// TwinCAT 3 PLC project TcLog
// Title: TcLog
// Company: Benedikt Geisler
// Author: Benedikt Geisler
// ProjectVersion: 0.6.1
// Description: TcLog provides logging functionality to TwinCAT.
// ProgramVersion: 3.1.4026.20
// libraries:
//   Tc2_Standard, * (Beckhoff Automation GmbH)
//   Tc2_System, * (Beckhoff Automation GmbH)
//   Tc2_Utilities, * (Beckhoff Automation GmbH)
//   Tc3_DynamicMemory, * (Beckhoff Automation GmbH)
// project tree:
//   / Constants.TcGVL (not stored)
//   Logger/DataTypes/ Error.TcDUT, ErrorCodes.TcDUT, LoggingConfiguration.TcDUT (not stored), LogLevels.TcDUT (not stored), RollingIntervals.TcDUT
//   Logger/Interfaces/ ILog.TcIO, ILogCore.TcIO
//   Logger/ LogLevelToAdsLogMsgType.TcPOU (not stored), TcLog.TcPOU (not stored), TcLogCore.TcPOU, TcLogTrig.TcPOU
//   StringBuilder/Interfaces/ ILimitedStringBuilder.TcIO (not stored), IStringBuilder.TcIO (not stored)
//   StringBuilder/ StringBuilder.TcPOU (not stored)
//   Utils/ AnyToString.TcPOU (not stored), DateTime.TcPOU, DeleteOldFiles.TcPOU (not stored), DynamicStringBuffer.TcPOU, GetFileAgeInSeconds.TcPOU (not stored)
//   Utils/DataTypes/ DeleteFilesState.TcDUT (not stored), PersistToFileState.TcDUT (not stored)

// ---- Logger/DataTypes/Error.TcDUT
/// This is the error type used in this library.
TYPE Error :
STRUCT
  /// `TRUE` signals an active error
	Active : BOOL;
  /// Error code of type `ErrorCodes`
	Code : INT;
  /// Plain text error message
	Info : Tc2_System.T_MaxString;
END_STRUCT
END_TYPE

// ---- Logger/DataTypes/ErrorCodes.TcDUT
/// Provides error codes for TcLogCore
{attribute 'qualified_only'}
{attribute 'strict'}
{attribute 'to_string'}
TYPE ErrorCodes : 
(
	None := 0,
	OpeningFileFailed,
	WritingToFileFailed,
	ClosingFileFailed,
	EnumeratingFilesInSpecifiedDirectoryFailed,
	DeletingFileFailed,
	FifoOverflow
);
END_TYPE

// ---- Logger/DataTypes/RollingIntervals.TcDUT
/// Rolling interval to create a new log file when expired. 
{attribute 'qualified_only'}
{attribute 'strict'}
{attrivute 'to_string'}
TYPE RollingIntervals :
(
	None := 0,
	Hourly,
	Daily,
	Monthly
);
END_TYPE

// ---- Logger/Interfaces/ILog.TcIO
INTERFACE PUBLIC ILog

METHOD SetLogger : BOOL
VAR_INPUT
    ref2Core : ILogCore;
END_VAR
END_METHOD

END_INTERFACE

// ---- Logger/Interfaces/ILogCore.TcIO
INTERFACE PUBLIC ILogCore EXTENDS __SYSTEM.IQueryInterface

// Logger method.
// Logs data in custom format. No additional formatting will be done.
METHOD LogCustomFormat : BOOL
VAR_INPUT
    data : Tc2_System.T_MaxString; // Data to be logged. No additional formatting will be done.
END_VAR
END_METHOD

// Logger method.
// Logs in the standard format. This includes
// - timestamp
// - log level
// - log message
// - instance path of logging source (optional)
// The message will only be logged if the logging level exceeds the configured minimum logging level.
METHOD LogStandardFormat : BOOL
VAR_INPUT
    data : Tc2_System.T_MaxString; // Data to be logged. Additional formatting wil be done.
    instancePath : Tc2_System.T_MaxString; // Instance path of calling logger to locate source of logging message.
    logLevel : LogLevels; // Log level of message.
END_VAR
END_METHOD

END_INTERFACE

// ---- Logger/TcLogCore.TcPOU
/// `TcLogCore` provides the base functionality of the logger and sets the configuration.
/// The logger can be configured by calling its methods that set the configuration.
///
/// > [!NOTE]
/// > `TcLogCore.RunLogger()` should be called once each cycle. The configuration methods should be called **before** 
/// > `RunLogger` is called.
///
/// When declaring an instance of TcLogCore, the ininital buffer size has to be set. If the buffer size is set too low, it will expand
/// automatically if enough memory is available.
///
/// To set the inital buffer size to accomodate 100 messages, use it like this:
///
/// ```st
/// VAR
///   myLogger: TcLogCore(BufferSize := 100 * (Tc2_System.MAX_STRING_LENGTH * Constants.FifoOverhead));
/// END_VAR
/// ```
///
{attribute 'linkalways'}
{attribute 'hide_all_locals'}
FUNCTION_BLOCK PUBLIC TcLogCore IMPLEMENTS ILogCore
VAR
	_loggingSingleton : TcLog; // Logger-Singleton: Required to provide Singleton-functionality for TcLog.
	_utcTimeAsFileTime : Tc2_Utilities.T_FILETIME; // Current utc time as filetime
	_localTimeAsSystemTime : Tc2_Utilities.TIMESTRUCT; // Current local time as timestring
	_localTimeAsString : STRING; // Current local time as string
	_logCache : DynamicStringBuffer; // Dynamic string buffer to cache logs to be processed
	_startLoggingConfiguration : BOOL; // Aux variable to provide fluent interface.
	_internalErrorOccured : BOOL; // Aux variable to log internal errors to Error-property.                                                   				
	_config : LoggingConfiguration; // Logging configuration. Is set by invoking configuration methods.
	_error : Error; // Contains information about internal error.
	_busy : BOOL; // Logger is busy, typically with writing logs to the file system.
  _timeInfoReady : BOOL := FALSE; // Set to true once the time information is available
END_VAR

// Nothing to be done here. Logger works by invoking its methods.
// "RunLogger" contains all the implementation that has to be processed cyclically.

// Builds logging configuration.
// Required to provide a fluent interface.
// Has to be called at the begin of each method that configures the logger.
{attribute 'hide'}
METHOD PRIVATE BuildLoggingConfiguration : BOOL
IF NOT _startLoggingConfiguration THEN
	_startLoggingConfiguration := TRUE;
	
	_config.RollingInterval := RollingIntervals.Daily;
	_config.WriteToAds := FALSE;
	_config.FileName := '';
	_config.FilePath := 'c:\';
	_config.MinimumLevel := LogLevels.Debug;
	_config.Delimiter := '|';
	_config.IncludeInstancePath := FALSE;
	_config.LogFileLifespan := 0;
	_config.TimestampFormat := 'YYYYMMDD_hhmm_';
	_config.ValidTimestampsOnly := FALSE;
END_IF
END_METHOD

/// `Busy` evaluates to `TRUE` as long as the log file is kept open to append new log messages
/// or there are pending messages in the queue to be written to the logfile.
{attribute 'monitoring':='call'}
PROPERTY Busy : BOOL
GET
Busy := _busy;
END_GET
SET // PRIVATE
_busy := Busy;
END_SET
END_PROPERTY

/// Returns the current configuration of the logger.
{attribute 'monitoring':='variable'}
PROPERTY Configuration : LoggingConfiguration
GET
Configuration := _config;
END_GET
END_PROPERTY

/// Configuration method which sets the lifespan of log files. Once exceeded, they will be deleted.
METHOD DeleteLogFilesAfterDays : REFERENCE TO TcLogCore
VAR_INPUT
  /// Lifespan of logfiles in days.
	lifespan : UINT; 
END_VAR
BuildLoggingConfiguration();

_config.LogFileLifespan := lifespan;

DeleteLogFilesAfterDays REF= THIS^;
END_METHOD

/// Returns information about internal errors.
{attribute 'monitoring':='call'}
{attribute 'suppress_wrn_C0410'}
PROPERTY Error : REFERENCE TO Error
GET
Error REF= _error;
END_GET
END_PROPERTY

METHOD FB_init : BOOL
VAR_INPUT
	bInitRetains : BOOL; // if TRUE, the retain variables are initialized (warm start / cold start)
	bInCopyCode : BOOL; // if TRUE, the instance afterwards gets moved into the copy code (online change)
  /// Initial buffer size for the internal log message buffer
	bufferSize : UDINT;
END_VAR
_loggingSingleton.Init(THIS^);
_logCache.Init(bufferSize);
END_METHOD

/// Flushes the logging cache. All messages that have not yet been processed will be lost.
METHOD FlushCache : BOOL
_logCache.FlushCache();
END_METHOD

/// Configuration method. If this method is called, the instance path where the log 
/// messages has been triggered will be included in the log message. 
METHOD IncludeInstancePath : REFERENCE TO TcLogCore
BuildLoggingConfiguration();

_config.IncludeInstancePath := TRUE;

IncludeInstancePath REF= This^;
END_METHOD

/// Logger method. It should only be called from within objects that implement `ILog`.
/// Logs data in custom format. No additional formatting will be done. 
METHOD LogCustomFormat : BOOL
VAR_INPUT
  /// Data to be logged.
	data : Tc2_System.T_MaxString; 
END_VAR
IF(TimeInfoReady OR NOT _config.ValidTimestampsOnly) THEN 
	IF _config.WriteToAds THEN 
		Tc2_System.ADSLOGSTR(ADSLOG_MSGTYPE_LOG OR ADSLOG_MSGTYPE_HINT, data, ''); 
	END_IF
	
	IF _config.FileName <> '' THEN 
		_logCache.AddLine(data);
	END_IF
END_IF
END_METHOD

/// Logger method. It should only be called from within objects that implement `ILog`.
/// Logs in the standard format. This includes
/// - timestamp
/// - log level
/// - log message
/// - instance path of logging source (optional)
/// The message will only be logged if the logging level exceeds the configured minimum logging level.
METHOD LogStandardFormat : BOOL
VAR_INPUT
  /// Data to be logged.
	data : Tc2_System.T_MaxString; 
  /// Instance path of calling logger to locate source of logging message.
	instancePath : Tc2_System.T_MaxString;
  /// Log level of message. 
	logLevel : LogLevels; 
END_VAR
VAR_INST
  {attribute 'hide'}
	messageBuilder : StringBuilder;
END_VAR
IF LogLevel >= _config.MinimumLevel AND (TimeInfoReady OR NOT _config.ValidTimestampsOnly)  THEN
	IF _config.WriteToAds THEN 
		Tc2_System.ADSLOGSTR(
			ADSLOG_MSGTYPE_LOG OR LogLevelToAdsLogMsgType(logLevel), 
			messageBuilder
				.Reset()
				.AppendIf(_config.IncludeInstancePath, instancePath)
				.AppendIf(_config.IncludeInstancePath, _config.Delimiter)
				.Append(data)
				.ToString(), 
			''
		); 
	END_IF
	
	IF _config.FileName <> '' THEN 
		_logCache.AddLine(
			messageBuilder
					.Reset()
					.Append(_localTimeAsString)
					.Append(_config.Delimiter)
					.Append(TO_STRING(LogLevel))
					.AppendIf(_config.IncludeInstancePath, _config.Delimiter)
					.AppendIf(_config.IncludeInstancePath, instancePath)
					.Append(_config.Delimiter)
					.Append(data)
					.ToString()
		);
	END_IF
END_IF
END_METHOD

/// Configuration method.
/// Sets the minimum log level. Log messages below this level 
/// will not be logged.
METHOD MinimumLevel : REFERENCE TO TcLogCore
VAR_INPUT
  /// Minimum log level to be logged.
	level : LogLevels; 
END_VAR
BuildLoggingConfiguration();

_config.MinimumLevel := level;

MinimumLevel REF=THIS^;
END_METHOD

// Checks the specified rolling interval for the file name.
// Generates new file name if rolling intervall exceeded.
{attribute 'hide_all_locals'}
{attribute 'hide'}
METHOD PRIVATE RollingIntervalReached : BOOL
VAR_INPUT
	currentUtcTime : Tc2_Utilities.TIMESTRUCT;  // Current system time as utc
	rollingInterval : RollingIntervals; // Rolling interval 
END_VAR
VAR_INST
	newHour : Tc2_Standard.R_TRIG;
	newDay : Tc2_Standard.R_TRIG;
	newMonth : Tc2_Standard.R_TRIG;
	
	hourRolled : BOOL;
	dayRolled : BOOL;
	monthRolled : BOOL;
END_VAR
newHour(CLK := (currentUtcTime.wMinute = 0 AND currentUtcTime.wSecond = 0), 
	Q => hourRolled);
newDay(CLK := (hourRolled AND currentUtcTime.wHour = 0), 
	Q => dayRolled);
newMonth(CLK := (dayRolled AND currentUtcTime.wDay = 1), 
	Q => monthRolled);

RollingIntervalReached := 	(hourRolled 	AND rollingInterval = RollingIntervals.Hourly) OR
							(dayRolled 		AND rollingInterval = RollingIntervals.Daily) 	OR
							(monthRolled 	AND rollingInterval = RollingIntervals.Monthly);
END_METHOD

/// Cyclic method of Logger.
/// This method has to be executed in every plc cycle and runs 
/// all internal methods that have to be executed cyclically.
/// > [!NOTE]
/// > This method should be the last method of `TcLogCore` to be called in each cycle.
{attribute 'hide_all_locals'}
METHOD RunLogger : BOOL
VAR_INST
	newDay : Tc2_Standard.R_TRIG; 
	dateTime : DateTime;
	deleteExpiredLogFiles : DeleteOldFiles;
	fileNameStringBuilder : StringBuilder;
	timeStamp : STRING; // Timestamp used for filename
END_VAR
// Generate time data (shared state)
dateTime();
IF dateTime.Done THEN _timeInfoReady := TRUE; END_IF

_localTimeAsSystemTime := dateTime.AsLocalSystemTime;
_localTimeAsString := dateTime.AsLocalSystemTimeString;
_utcTimeAsFileTime := dateTime.AsUtcFileTime;

// Generate new timestamp for filename
IF RollingIntervalReached(_localTimeAsSystemTime, _config.RollingInterval) OR dateTime.Done THEN
	timeStamp := dateTime.ToFormatString(_config.TimestampFormat);
END_IF

// Delete expired log files
newDay(CLK := _localTimeAsSystemTime.wHour = 0);
deleteExpiredLogFiles(
	StartScan 			:= 	newDay.Q AND (_config.LogFileLifespan > 0),
	ExpirationInDays 	:=	_config.LogFileLifespan,
	FilePath			:=	_config.FilePath,
	FileName 			:=	_config.FileName,
	CurrentUtcTime 		:= 	_utcTimeAsFileTime	
	);
IF deleteExpiredLogFiles.Error.Active THEN
	_internalErrorOccured := TRUE;
	_error := deleteExpiredLogFiles.Error;
END_IF
		
// Persist logging messages to file
_logCache.PersistToFile(
  TimeInfoReady,
	fileNameStringBuilder
		.Reset()
		.Append(_config.FilePath)
		.AppendIf(Tc2_Standard.RIGHT(_config.FilePath, 1) <> '\', '\')
		.Append(timeStamp)
		.Append(_config.FileName)
		.ToString()
);
IF _logCache.Error.Active THEN
	_internalErrorOccured := TRUE;
	_error := _logCache.Error;
END_IF

// Forward busy state of LogCache 
Busy := _logCache.Busy;

// Reset Logging configuration: neccesary in order to provide fluent interface
_startLoggingConfiguration := FALSE;

// Reset error flag each cycle to automatically confirm errors once they are gone.
IF NOT _internalErrorOccured THEN
	_error.Active := FALSE;
	_error.Code := ErrorCodes.None;
	_error.Info := '';
END_IF
_internalErrorOccured := FALSE;
END_METHOD

/// Configuration method
/// Sets delimiter between different columns of log file.
METHOD SetDelimiter : REFERENCE TO TcLogCore
VAR_INPUT
  /// Delimiter between different columns of log file.
	delimiter : STRING(1); 
END_VAR
BuildLoggingConfiguration();

_config.Delimiter := delimiter;

SetDelimiter REF=THIS^;
END_METHOD

/// Configuration method.
/// Sets the rolling interval of the log file. Once the rolling interval
/// expires, a file name with a new timestamp will be generated.
METHOD SetRollingInterval : REFERENCE TO TcLogCore
VAR_INPUT
  /// Rolling interval for log file. Once exceeded, a new log file will be created.
	interval : RollingIntervals; 
END_VAR
BuildLoggingConfiguration();

_config.RollingInterval := interval;

SetRollingInterval REF= THIS^;
END_METHOD

/// `TimeInfoReady` evaluates to `TRUE` once the time information used by determine
/// the timestamp for the message is available.
{attribute 'monitoring':='call'}
PROPERTY TimeInfoReady : BOOL
GET
TimeInfoReady := _timeInfoReady;
END_GET
END_PROPERTY

/// Configuration method.
/// Sets the format of the timestamp in the file name. 
/// 
/// The following format options are available:
///	Y : year
///	M : month
/// D : day
/// h : hour 
/// m : minute
/// s : second
/// i : millisecond
/// 
/// Example: _YYMMDD-hh:mm:ss:iii_
/// => _20210812-12:30:22:123_
METHOD TimestampFormat : REFERENCE TO TcLogCore
VAR_INPUT
  /// Format the timestamp should have.
	format : STRING; 
END_VAR
BuildLoggingConfiguration();

_config.TimestampFormat := format;

TimestampFormat REF= THIS^;
END_METHOD

/// Configuration method. If this method is called, only valid timestamps are logged.
/// Note that using this configuration will skip logging anything during the first few PLC cycles, 
/// as TwinCAT needs a few cycles to initialize its time information.
METHOD ValidTimestampsOnly : REFERENCE TO TcLogCore
BuildLoggingConfiguration();

_config.ValidTimestampsOnly := TRUE;

ValidTimestampsOnly REF= This^;
END_METHOD

/// Configuration method.
/// If this method is called, the logs will be written to ADS.
METHOD WriteToAds : REFERENCE TO TcLogCore
BuildLoggingConfiguration();

_config.WriteToAds := TRUE;

WriteToAds REF= This^;
END_METHOD

/// Configuration method.
/// If this method is called, the logs will be persisted to the file system.
METHOD WriteToFile : REFERENCE TO TcLogCore
VAR_INPUT
  /// File path the logs will be written to.
	path : Tc2_System.T_MaxString; 
  /// File name of the log file. Will automatically be prefixed by timestamp.
	fileName : STRING; 
END_VAR
BuildLoggingConfiguration();

IF Tc2_Standard.RIGHT(path, 1) <> '\' THEN
  _config.FilePath := TC2_Standard.CONCAT(path, '\');  
ELSE
  _config.FilePath := path;
END_IF
_config.FileName := fileName;

WriteToFile REF= This^;
END_METHOD

END_FUNCTION_BLOCK

// ---- Utils/DynamicStringBuffer.TcPOU
{attribute 'hide_all_locals'}
FUNCTION_BLOCK INTERNAL DynamicStringBuffer
VAR_OUTPUT
  Error : Error; // Error information of this FB
END_VAR
VAR
  _fifo : Tc2_Utilities.FB_StringRingBuffer; // Necessary to buffer log data until it has been written to file.
  _memoryManager : Tc3_DynamicMemory.FB_DynMem_Manager; // Memory manager, required by DynMem_Buffer.
  _dynamicMemoryBuffer : Tc3_DynamicMemory.FB_DynMem_Buffer(ipMemMan := _memoryManager); // Provides dynamic buffer for Fifo. Is extended automatically if more than the
                                                                   // default buffer size is needed.                  
  _busy : BOOL; // Buffer is busy; typically with writing data to the file system.
END_VAR

METHOD AddLine : BOOL
VAR_INPUT
  text : Tc2_System.T_MaxString; // Text to be added to the buffer
END_VAR
ResizeFifoBufferIfNecessary();
_fifo.A_AddTail(putValue := Tc2_Standard.CONCAT(Tc2_Standard.LEFT(text, 254), '$N'));
END_METHOD

METHOD AddString : BOOL
VAR_INPUT
  text : Tc2_System.T_MaxString; // String to be added to the buffer
END_VAR
ResizeFifoBufferIfNecessary();
_fifo.A_AddTail(putValue := text);
END_METHOD

METHOD PRIVATE AllocateBuffer : BOOL // Allocates buffer FOR the fifo.
VAR_INPUT
  bufferSize : UDINT; // Initial buffer size in BYTEs for fifo buffer.
END_VAR
_dynamicMemoryBuffer.CreateBuffer(nSize:=bufferSize, bReset:=TRUE);
_fifo.pBuffer := _dynamicMemoryBuffer.pBuffer;
_fifo.cbBuffer := bufferSize;
END_METHOD

{attribute 'monitoring':='call'}
PROPERTY Busy : BOOL
GET
Busy := _busy;
END_GET
SET // PRIVATE
_busy := Busy;
END_SET
END_PROPERTY

METHOD FB_exit : BOOL
VAR_INPUT
  bInCopyCode : BOOL; // if TRUE, the exit method is called for exiting an instance that is copied afterwards (online change).
END_VAR
_dynamicMemoryBuffer.Clear();
END_METHOD

METHOD FlushCache : BOOL
_fifo.A_Reset();
END_METHOD

METHOD INTERNAL Init : BOOL
VAR_INPUT
  bufferSize : UDINT; // Initial buffer size in BYTEs for fifo buffer.
END_VAR
AllocateBuffer(bufferSize);
END_METHOD

{attribute 'hide_all_locals'}
METHOD PersistToFile : BOOL
VAR_INPUT
  enable: BOOL; // TRUE starts persistence mechanism
  fileName : Tc2_System.T_MaxString; // File name including its path
END_VAR
VAR_INST
  state : PersistToFileState;
  
  fileOpen : Tc2_System.FB_FileOpen;
  fileHandle : UINT;
  
  fileWrite : Tc2_System.FB_FileWrite;
  lockFileWriteToForceRisingEdge : BOOL; // filePuts can only be executed every other cycle
                                         // since it needs a rising edge to execute.
  fileClose : Tc2_System.FB_FileClose;
  
  buffer : ARRAY[0..CONSTANTS.BufferSize] OF BYTE;
  currentBufferPos : UDINT;
  fifoHeadString : Tc2_System.T_MaxString;
  fifoHeadLength : UDINT;
  fifoHeadBytes : ARRAY[0..Tc2_System.MAX_STRING_LENGTH] OF BYTE;
  i : UINT;
END_VAR
VAR CONSTANT
  NetId : STRING := '';
  Timeout : TIME := DEFAULT_ADS_TIMEOUT;
  MaxLogsPerCycle : UINT := UDINT_TO_UINT(CONSTANTS.BufferSize / Tc2_System.MAX_STRING_LENGTH);
  MaxBufferPosition : UDINT := (SIZEOF(buffer)-Tc2_System.MAX_STRING_LENGTH);
END_VAR
// State machine
// Using if-statements instead of case for performance reasons:
// Some states execute instantly and allow thus the next state 
// to start within the same plc cycle.

// *** I D L E ***
IF state = PersistToFileState.Idle THEN
  lockFileWriteToForceRisingEdge := FALSE;
  IF _fifo.nCount > 0 AND enable THEN 
    lockFileWriteToForceRisingEdge := FALSE;
    state := PersistToFileState.OpenFile;
  END_IF
END_IF
    
// *** O P E N   F I L E ***
fileOpen(sNetId := NetId, sPathName := fileName, nMode := FOPEN_MODEAPPEND OR FOPEN_MODETEXT, 
           ePath := PATH_GENERIC, bExecute := (state = PersistToFileState.OpenFile), tTimeout := Timeout,
           hFile => fileHandle);

IF state = PersistToFileState.OpenFile THEN
  IF fileOpen.bError THEN
    state := PersistToFileState.CloseFile;
  ELSIF NOT fileOpen.bBusy THEN
    state := PersistToFileState.GetStringFromFifo; 
  END_IF
END_IF 

// *** P O P   F R O M   F I F O ***
IF state = PersistToFileState.GetStringFromFifo THEN
  IF NOT lockFileWriteToForceRisingEdge THEN
    currentBufferPos := 0;
    FOR i:=0 TO MaxLogsPerCycle DO
      IF _fifo.nCount <= 0 THEN EXIT; END_IF
      IF currentBufferPos >= MaxBufferPosition THEN EXIT; END_IF
      
      _fifo.A_RemoveHead(getValue => fifoHeadString); 
      fifoHeadBytes := MAXSTRING_TO_BYTEARR(fifoHeadString);
      fifoHeadLength := INT_TO_UDINT(LEN(fifoHeadString));
      MEMCPY(
        destAddr  :=  ADR(buffer) + SIZEOF(BYTE) * currentBufferPos,
        srcAddr   :=  ADR(fifoHeadBytes),
        n     :=  fifoHeadLength);    
      currentBufferPos := currentBufferPos + fifoHeadLength;  
    END_FOR
    state := PersistToFileState.AppendDataToFile;
  END_IF
  lockFileWriteToForceRisingEdge := FALSE;
END_IF
  
// *** W R I T E   T O   F I L E ***
fileWrite(
  sNetId := NetId, 
  hFile := fileHandle, 
  pWriteBuff := ADR(buffer),
  cbWriteLen := currentBufferPos,
  bExecute := state = PersistToFileState.AppendDataToFile, 
  tTimeout := Timeout); 

IF state = PersistToFileState.AppendDataToFile THEN
  lockFileWriteToForceRisingEdge := TRUE;   
  IF fileWrite.bError THEN
    state := PersistToFileState.CloseFile;
  ELSIF _fifo.nCount > 0 AND NOT fileWrite.bBusy THEN
    state := PersistToFileState.GetStringFromFifo; 
  ELSIF _fifo.nCount = 0 THEN
    state := PersistToFileState.CloseFile;
  END_IF
END_IF
    
// *** C L O S E   F I L E ***
fileClose(
  sNetId := NetId, hFile := fileHandle, 
  bExecute := (state = PersistToFileState.CloseFile), tTimeout := Timeout);

IF state = PersistToFileState.CloseFile THEN
  IF NOT fileClose.bBusy THEN state := PersistToFileState.Idle; END_IF
END_IF

// Close file in case of error
IF fileOpen.bError THEN state := PersistToFileState.CloseFile; END_IF
IF fileWrite.bError THEN state := PersistToFileState.CloseFile; END_IF
IF NOT _fifo.bOk AND _fifo.nCount > 0 AND state <> PersistToFileState.Idle THEN 
  state := PersistToFileState.CloseFile; 
END_IF

// Error handling
IF fileOpen.bError THEN
  Error.Active := TRUE;
  Error.Code := ErrorCodes.OpeningFileFailed;
  Error.Info := Tc2_Standard.CONCAT('Opening file failed. Error thrown by FB_FileOpen. Consult Beckhoff InfoSys. Internal Error: ', UDINT_TO_STRING(fileOpen.nErrId));
ELSIF fileWrite.bError THEN
  Error.Active := TRUE;
  Error.Code := ErrorCodes.WritingToFileFailed;
  Error.Info := Tc2_Standard.CONCAT('Writing to file failed. Error thrown by FB_FileWrite. Consult Beckhoff InfoSys. Internal Error: ', UDINT_TO_STRING(fileWrite.nErrId));
ELSIF fileClose.bError THEN
  Error.Active := TRUE;
  Error.Code := ErrorCodes.ClosingFileFailed;
  Error.Info := Tc2_Standard.CONCAT('Closing file failed. Error thrown by FB_FileClose. Consult Beckhoff InfoSys. Internal Error: ', UDINT_TO_STRING(fileClose.nErrId));
ELSIF NOT _fifo.bOk AND _fifo.nCount > 0 THEN
  Error.Active := TRUE;
  Error.Code := ErrorCodes.FifoOverflow;
  Error.Info := 'FIFO overflow. Check if plc has enough free memory.';
ELSE
  Error.Active := FALSE;
  Error.Code := ErrorCodes.None;
  Error.Info := '';
END_IF

// Set busy state
Busy := (state <> PersistToFileState.Idle OR _fifo.nCount > 0);

(* Uncomment for cyclic logging of state machine, buffer usage & errors

ADSLOGSTR(ADSLOG_MSGTYPE_LOG, 
  Tc2_Standard.CONCAT('****DynamicStringBuffer.state:', 
  Tc2_Standard.CONCAT(UINT_TO_STRING(state),
  Tc2_Standard.CONCAT(', DynamicStringBuffer.hFile:', UINT_TO_STRING(hFile)))), '');

ADSLOGSTR(ADSLOG_MSGTYPE_LOG, 
  Tc2_Standard.CONCAT('****Fifo: used ', 
  Tc2_Standard.CONCAT(UDINT_TO_STRING(Fifo.cbSize),
  Tc2_Standard.CONCAT(' of ', UDINT_TO_STRING(Fifo.cbBuffer)))), '');
  
IF Error.Active THEN
  ADSLOGSTR(ADSLOG_MSGTYPE_LOG, 
    Tc2_Standard.CONCAT('****DynamicStringBuffer.Error: ', Error.Info), 
    '');  
END_IF
*)
END_METHOD

METHOD PopHead : Tc2_System.T_MaxString
VAR_INST
  headString : Tc2_System.T_MaxString;
END_VAR
_fifo.A_RemoveHead(getValue => headString);
PopHead := headString;
END_METHOD

// Resizes the buffer for the FIFO if necessary
METHOD PRIVATE ResizeFifoBufferIfNecessary : BOOL
VAR
  requiredSize : UDINT;
  newSize : DINT;
END_VAR
requiredSize := _fifo.cbSize + (Tc2_System.MAX_STRING_LENGTH + Constants.FifoOverhead);

IF requiredSize > _fifo.cbBuffer THEN
  _dynamicMemoryBuffer.Resize(nSize := requiredSize*SIZEOF(BYTE), bPreserve:=TRUE, bReset:=TRUE);
  _fifo.pBuffer := _dynamicMemoryBuffer.pBuffer;
  _fifo.cbBuffer := requiredSize;
END_IF
END_METHOD

END_FUNCTION_BLOCK

// ---- Utils/DateTime.TcPOU
/// Generate time data in different formats.
{attribute: 'hide_all_locals'}
FUNCTION_BLOCK DateTime
VAR
  _localSystemTime : Tc2_Utilities.FB_LocalSystemTime;
  _getSystemTime : Tc2_System.GETSYSTEMTIME;
  _timeZoneInfo : Tc2_Utilities.FB_GetTimeZoneInformation;
  _localTime : Tc2_Utilities.FB_SystemTimeToTzSpecificLocalTime;
  _localSystemTimeValid : Tc2_Standard.R_TRIG;
  _utcTime : Tc2_Utilities.FB_TzSpecificLocalTimeToFileTime;
END_VAR

// Get local system time
_localSystemTime(
  sNetID  :=  '',
  bEnable :=  TRUE,
  dwCycle :=  1,
  dwOpt :=  1,
  tTimeout:=  DEFAULT_ADS_TIMEOUT
);

// Get timezone information
_timeZoneInfo(
  sNetID := '',
  bExecute := TRUE,
  tTimeout := DEFAULT_ADS_TIMEOUT);

// Convert local time to utc time
_utcTime(
  in := THIS^.AsLocalFileTime,
  tzInfo := _timeZoneInfo.tzInfo);
  
// Finished retrieving time data
_localSystemTimeValid(CLK := _localSystemTime.bValid);

/// Returns local time as `Tc2_Utilities.T_FILETIME`.
{attribute 'monitoring':='variable'}
PROPERTY AsLocalFileTime : Tc2_Utilities.T_FILETIME
GET
AsLocalFileTime := SYSTEMTIME_TO_FILETIME(THIS^.AsLocalSystemTime);
END_GET
END_PROPERTY

/// Returns local time as `Tc2_Utilities.TIMESTRUCT`.
{attribute 'monitoring':='variable'}
PROPERTY AsLocalSystemTime : Tc2_Utilities.TIMESTRUCT
GET
AsLocalSystemTime := _localSystemTime.systemTime;
END_GET
END_PROPERTY

/// Returns local time as string.
{attribute 'monitoring':='variable'}
PROPERTY AsLocalSystemTimeString : Tc2_System.T_MAXSTRING
GET
AsLocalSystemTimeString := Tc2_Utilities.SYSTEMTIME_TO_STRING(THIS^.AsLocalSystemTime);
END_GET
END_PROPERTY

/// Returns UTC time as `Tc2_Utilities.T_FILETIME`.
{attribute 'monitoring':='variable'}
PROPERTY AsUtcFileTime : Tc2_Utilities.T_FILETIME
GET
AsUtcFileTime := _utcTime.out;
END_GET
END_PROPERTY

/// When calling `DateTime` the first time, it takes some time until all time and timezone information is available.
/// `Done` is `TRUE` for one cycle, once all the data is ready. 
{attribute 'monitoring':='call'}
PROPERTY Done : BOOL
GET
Done := _localSystemTimeValid.Q;
END_GET
END_PROPERTY

// Replaces placeholders in format string by the actual time values.
{attribute 'hide_all_locals'}
{attribute 'hide'}
METHOD PRIVATE ReplaceFormatPlaceholder : STRING
VAR_INPUT
  format : STRING;
  length : INT;
  timeType : STRING(1);
END_VAR
VAR_INST
  i : INT;
  replaceString : STRING;
  timeString : STRING;
END_VAR
VAR
  localSystemTime : Tc2_Utilities.TIMESTRUCT;
END_VAR
localSystemTime := THIS^.AsLocalSystemTime;

IF    timeType = 'Y'  THEN timeString := TO_STRING(localSystemTime.wYear); 
ELSIF timeType = 'M'  THEN timeString := TO_STRING(localSystemTime.wMonth); 
ELSIF timeType = 'D'  THEN timeString := TO_STRING(localSystemTime.wDay); 
ELSIF timeType = 'h'  THEN timeString := TO_STRING(localSystemTime.wHour); 
ELSIF timeType = 'm'  THEN timeString := TO_STRING(localSystemTime.wMinute); 
ELSIF timeType = 's'  THEN timeString := TO_STRING(localSystemTime.wSecond); 
ELSIF timeType = 'i'  THEN timeString := TO_STRING(localSystemTime.wMilliseconds); 
ELSE
  timeString:='';
END_IF

replaceString := '';

IF length > Tc2_Standard.LEN(timeString) THEN
  FOR i:=1 TO length - Tc2_Standard.LEN(timeString) DO
    replaceString := Tc2_Standard.CONCAT(replaceString, '0');
  END_FOR
  replaceString := Tc2_Standard.CONCAT(replaceString, timeString);
ELSE
  replaceString := Tc2_Standard.RIGHT(timeString, length);
END_IF

ReplaceFormatPlaceholder := Tc2_Standard.REPLACE(format, replaceString, length, Tc2_Standard.FIND(format, timeType));
END_METHOD

/// Returns a formatted string containing the actual time information 
/// - `Y` : year
/// - `M` : month
/// - `D` : day
/// - `h` : hour 
/// - `m` : minute
/// - `s` : second
/// - `i` : millisecond
/// 
/// Example:    
/// _YYMMDD-hh:mm:ss:iii_   
/// => _20210812-12:30:22:123_
{attribute 'hide_all_locals'}
METHOD ToFormatString : Tc2_System.T_MaxString
VAR_INPUT
  /// Format the timestamp should have.
  format : STRING;
END_VAR
VAR_INST
  inputString : STRING;
  c : STRING(1);
  formattedString : Tc2_System.T_MaxString;
END_VAR
VAR
  year : INT := 0;
  month : INT := 0;
  day : INT := 0;
  hour : INT := 0;
  minute : INT := 0;
  second : INT := 0;
  millisecond : INT := 0;
END_VAR
VAR CONSTANT
  ValidFormat : STRING := 'YMDhms';
END_VAR
// Parses "format" and returns a adequatly formatted string containing the time information
inputString := format;

WHILE Tc2_Standard.LEN(inputString) > 0 DO
  c := Tc2_Standard.LEFT(inputString, 1);
  
  IF    c = 'Y' THEN year := year + 1;
  ELSIF c = 'M' THEN month := month + 1;
  ELSIF c = 'D' THEN day := day + 1;
  ELSIF c = 'h' THEN hour := hour + 1;
  ELSIF c = 'm' THEN minute := minute + 1;
  ELSIF c = 's' THEN second := second + 1;
  ELSIF c = 'i' THEN millisecond := millisecond + 1;
  END_IF
  
  inputString := Tc2_Standard.DELETE(inputString, 1, 1);
END_WHILE

formattedString := ReplaceFormatPlaceholder(format, year, 'Y');
formattedString := ReplaceFormatPlaceholder(formattedString, month, 'M');
formattedString := ReplaceFormatPlaceholder(formattedString, day, 'D');
formattedString := ReplaceFormatPlaceholder(formattedString, hour, 'h');
formattedString := ReplaceFormatPlaceholder(formattedString, minute, 'm');
formattedString := ReplaceFormatPlaceholder(formattedString, second, 's');
formattedString := ReplaceFormatPlaceholder(formattedString, millisecond, 'i');

ToFormatString := formattedString;
END_METHOD

END_FUNCTION_BLOCK

// ---- Logger/TcLogTrig.TcPOU
/// This function block can be used to log on rising or falling edges.
/// For each signal that should be watched, a separate instance of `TcLogTrig` 
/// must be created.
{attribute 'linkalways'}
FUNCTION_BLOCK PUBLIC TcLogTrig EXTENDS TcLog

/// Logs data on falling edge of `CLK`.
{attribute 'hide_all_locals'}
METHOD OnFallingEdge : REFERENCE TO TcLog
VAR_INPUT
  /// Falling edge triggers logging the data.
  CLK : BOOL; 
END_VAR
VAR_INST
    fTrig : Tc2_Standard.F_TRIG;
END_VAR
fTrig(CLK:=CLK);

SUPER^.OnCondition(fTrig.Q);

OnFallingEdge REF= THIS^;
END_METHOD

/// Logs data on rising edge of `CLK`.
{attribute 'hide_all_locals'}
METHOD OnRisingEdge : REFERENCE TO TcLog
VAR_INPUT
  /// Rising edge logs data.
  CLK : BOOL; 
END_VAR
VAR_INST
    rTrig : Tc2_Standard.R_TRIG;
END_VAR
rTrig(CLK:=CLK);

SUPER^.OnCondition(rTrig.Q);

OnRisingEdge REF= THIS^;
END_METHOD

END_FUNCTION_BLOCK
